// TwinCAT 3 PLC project ConveyorBelt
// ProgramVersion: 3.1.4022.3
// libraries:
//   Tc2_Standard, * (Beckhoff Automation GmbH)
//   Tc2_System, * (Beckhoff Automation GmbH)
//   Tc3_Module, * (Beckhoff Automation GmbH)
//   VisuSymbols,3.5.10.0,System
// project tree:
//   / GlobalTextList.TcGTLO, PlcTask.TcTTO, Visualization Manager.TcVMO (not stored)
//   POUs/ MAIN.TcPOU
//   VISUs/ Visualization.TcVIS
// real-time tasks:
//   TASK PlcTask: cycle T#10ms, priority 20, ADS port 350

CONFIGURATION ConveyorBelt
    RESOURCE PLC ON TwinCAT3
        TASK PlcTask(INTERVAL := T#10ms, PRIORITY := 20);
        PROGRAM MAIN WITH PlcTask : MAIN;
    END_RESOURCE
END_CONFIGURATION

// ---- POUs/MAIN.TcPOU
PROGRAM MAIN
VAR
	start: BOOL;
	stop: BOOL;
	
	step1: RS;
	step2: RS;
	step3: RS;
	step4: RS;
	step5: RS;
	step6: RS;
	timer1: TON;
END_VAR


VAR_INPUT
	// Elevator inputs
	ElevatorSensor AT %IX1.0: BOOL; // Sensor attached to elevator
	ElevatorTableIsLifted AT %IX1.1: BOOL; // Elevator is currently lifted
	ElevatorTableIsDescended AT %IX1.2: BOOL; // Elevator is currently descended
	
	// Conveyor 2 inputs
	Conveyor2Sensor AT %IX2.0: BOOL; // Sensor attached to second conveyor
	PusherPushed AT %IX2.1: BOOL; // Pusher is pushed
	PusherRetracted AT %IX2.2: BOOL; // Pusher is retracted
END_VAR

VAR_OUTPUT
	// Conveyor 1 outputs
	Conveyor1 AT %QX0.0: BOOL; // First conveyor on/off
	
	// Elevator outputs
	ElevatorConveyor AT %QX1.0: BOOL; // Elevator's conveyor on/off
	ElevatorTableUp AT %QX1.1: BOOL; // Move elevator's table up
	ElevatorTableDown AT %QX1.2: BOOL; // Move elevator's table down
	
	// Conveyor 2 outputs
	Conveyor2 AT %QX2.0: BOOL; // Second conveyor on/off
	PusherPush AT %QX2.1: BOOL; // Push with pusher
	PusherRetract AT %QX2.2: BOOL; // Retract pusher
	
	// Box outputs
	BoxShaker AT %QX3.0: BOOL; // Shake the box
END_VAR

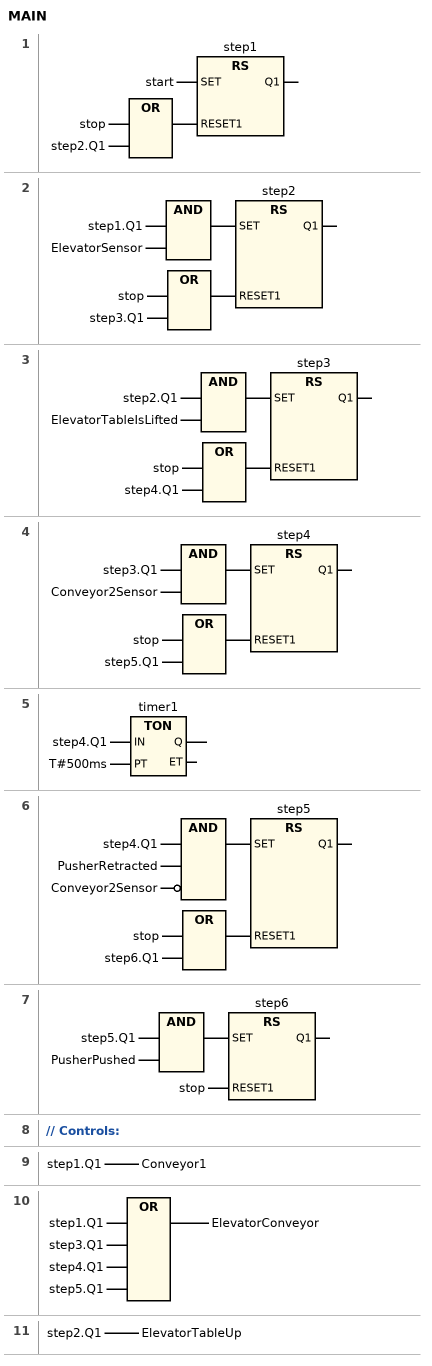
// NETWORK 1
step1(SET := start, RESET1 := stop OR step2.Q1); // RS

// NETWORK 2
step2(SET := step1.Q1 AND ElevatorSensor, RESET1 := stop OR step3.Q1); // RS

// NETWORK 3
step3(SET := step2.Q1 AND ElevatorTableIsLifted, RESET1 := stop OR step4.Q1); // RS

// NETWORK 4
step4(SET := step3.Q1 AND Conveyor2Sensor, RESET1 := stop OR step5.Q1); // RS

// NETWORK 5
timer1(IN := step4.Q1, PT := T#500ms); // TON

// NETWORK 6
step5(SET := step4.Q1 AND PusherRetracted AND NOT Conveyor2Sensor, RESET1 := stop OR step6.Q1); // RS

// NETWORK 7
step6(SET := step5.Q1 AND PusherPushed, RESET1 := stop); // RS

// NETWORK 8
// label: // Controls

// NETWORK 9
Conveyor1 := step1.Q1;

// NETWORK 10
ElevatorConveyor := step1.Q1 OR step3.Q1 OR step4.Q1 OR step5.Q1;

// NETWORK 11
ElevatorTableUp := step2.Q1;

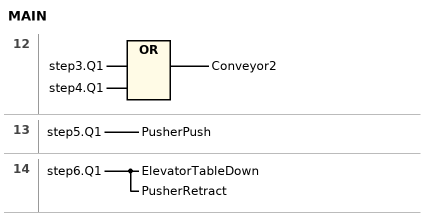
// NETWORK 12
Conveyor2 := step3.Q1 OR step4.Q1;

// NETWORK 13
PusherPush := step5.Q1;

// NETWORK 14
ElevatorTableDown := step6.Q1;
PusherRetract := step6.Q1;

END_PROGRAM

// ---- GlobalTextList.TcGTLO
TEXTLIST GlobalTextList
  854 = 'Conveyor 1'
  240 = 'Conveyor 2'
  266 = 'Conveyor 2 sensor'
  474 = 'Elevator Conveyor'
  698 = 'Elevator lifted'
  995 = 'Elevator sensor'
  175 = 'Elevator table descended'
  895 = 'Elevator table lifted'
  497 = 'Elevator table up'
  529 = 'Pusher pushed'
  615 = 'Pusher retracted'
END_TEXTLIST

// ---- VISUs/Visualization.TcVIS
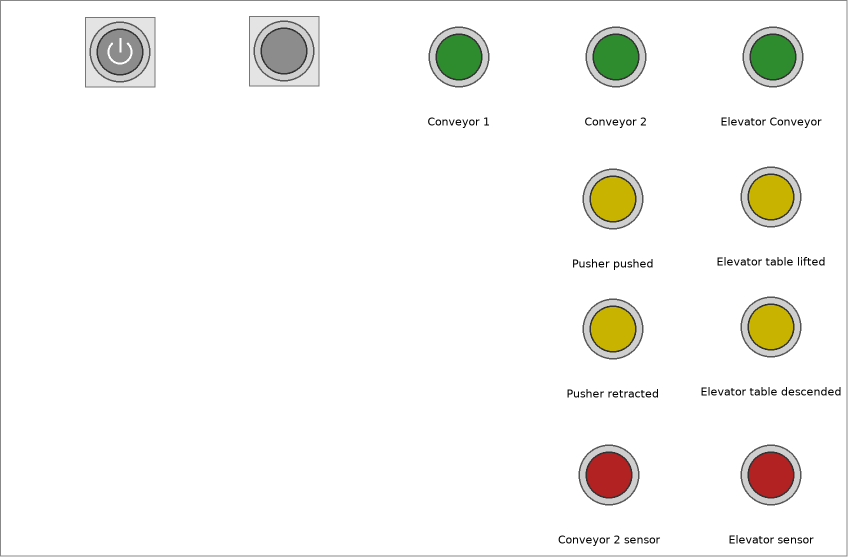
VISUALIZATION Visualization  // 848x557
    PowerSwitch (85,17 70x70), variable: MAIN.start, behaviour: TAP, style: Switch-PowerSwitch-Gray
    PushSwitch (249,16 70x70), variable: MAIN.stop, behaviour: TAP, style: Switch-PushSwitch-Gray
    Lamp1 (424,22 70x70), variable: MAIN.Conveyor1, style: Lamp-Lamp1-Green
    Label (384,107 150x30), "Conveyor 1"
    Lamp1 (581,22 70x70), variable: MAIN.Conveyor2, style: Lamp-Lamp1-Green
    Label (541,107 150x30), "Conveyor 2"
    Lamp1 (738,22 70x70), variable: MAIN.ElevatorConveyor, style: Lamp-Lamp1-Green
    Label (696,107 150x30), "Elevator Conveyor"
    Lamp1 (736,162 70x70), variable: MAIN.ElevatorTableIsLifted, style: Lamp-Lamp1-Yellow
    Label (696,247 150x30), "Elevator table lifted"
    Lamp1 (736,292 70x70), variable: MAIN.ElevatorTableIsDescended, style: Lamp-Lamp1-Yellow
    Label (696,377 150x30), "Elevator table descended"
    Lamp1 (736,440 70x70), variable: MAIN.ElevatorSensor, style: Lamp-Lamp1-Red
    Label (696,525 150x30), "Elevator sensor"
    Lamp1 (578,164 70x70), variable: MAIN.PusherPushed, style: Lamp-Lamp1-Yellow
    Label (538,249 150x30), "Pusher pushed"
    Lamp1 (578,294 70x70), variable: MAIN.PusherRetracted, style: Lamp-Lamp1-Yellow
    Label (538,379 150x30), "Pusher retracted"
    Lamp1 (574,440 70x70), variable: MAIN.Conveyor2Sensor, style: Lamp-Lamp1-Red
    Label (534,525 150x30), "Conveyor 2 sensor"
END_VISUALIZATION
